// TIA Portal V17 export
// export: Created 2025-06-26T06:49:26.9154109Z, ExportSetting WithDefaults, DisplayName Totally Integrated Automation Portal, DisplayVersion V17 Update 8, DisplayName TIA Portal Openness, DisplayVersion V17 Update 8, DisplayName TIA Portal Version Control Interface, DisplayVersion V17, DisplayName STEP 7 Professional, DisplayVersion V17 Update 8, DisplayName STEP 7 Safety, DisplayVersion V17 Update 6, DisplayName WinCC Advanced, DisplayVersion V17 Update 8
TYPE "stRegulatingValve"
// stored: IsFailsafeCompliant false
   STRUCT
      Cmd : Struct
         bManualMode : Bool;   // 1 = Manual Mode
         fManualValue : Real;   // manual position
         fOffset : Real;   // zero position offset
         Position : "stAnalogOutput";
      END_STRUCT;
      Stat : Struct
         Position : "stAnalogInput";
      END_STRUCT;
   END_STRUCT;
END_TYPE
